(* CODESYS project TONR.library
   Company: refik.com.tr
   DefaultNamespace: TONR
   Title: TONR
   Description: Kalıcı TON Timer
   Author: refik
   Version: 1.0

Project tree, tasks and I/O mapping:
  function block TONR [ST]
*)

// TONR
FUNCTION_BLOCK TONR
VAR_INPUT
	IN			: 		BOOL;
	PT			: 		TIME;
	TimeReset	: 		BOOL;
END_VAR
VAR_OUTPUT
	Current_ET	: 		TIME;	
	Total_ET	: 		TIME;
	RT			: 		TIME;
	Q			: 		BOOL;
END_VAR
VAR
	TON_Timer	: 		TON;
	SetPT		: 		TIME;
	mPT			: 		TIME;
	
	
END_VAR

//refik.com.tr

TON_Timer();TON_Timer.IN:=IN;Current_ET:=TON_Timer.ET;Total_ET:=mPT-RT;RT:=(TON_Timer.PT-TON_Timer.ET);Q:=(TON_Timer.Q);setPT:=SEL(IN,SetPT,RT);
IF PT=SetPT THEN mPT:=PT; END_IF
IF NOT IN AND (mPT<>PT) OR TimeReset THEN SetPT:=PT; END_IF
IF NOT IN THEN TON_Timer.PT:=SetPT; END_IF
//refik.com.tr

END_FUNCTION_BLOCK
